TYPE Type_CommIn_Conveyor :
STRUCT
	s_Robot			:Type_ModuleCommIn_Conveyor;
END_STRUCT
END_TYPE

(* stored: Version 1.1.0.1, ProductVersion 3.1.4024.9
   DUT Type_CommIn_Conveyor: Id {587db6c3-df60-4630-80e2-75fc91558d24} *)
